// TIA Portal V18 export
DATA_BLOCK "Motor control function FB_DB"   // DB1
VERSION : 0.1
// stored: AutoNumber true, DBAccessibleFromOPCUA true, InstanceOfName Motor control function FB, InstanceOfType FB
"Motor control function FB"
   // VAR_INPUT
   //    "FB Start" : Bool;
   //    "FB Stop" : Bool;
   //    "FB CB Feedback" : Bool;
   // END_VAR
   // VAR_OUTPUT
   //    "FB Motor contactor" : Bool;
   // END_VAR
BEGIN
END_DATA_BLOCK
